PROGRAM progFCVCntrl
VAR
	FCV_04_0100 : fbFCV;
	FCV_04_1001 : fbFCV;
	FCV_04_1002 : fbFCV;
	FCV_04_1003 : fbFCV;
END_VAR

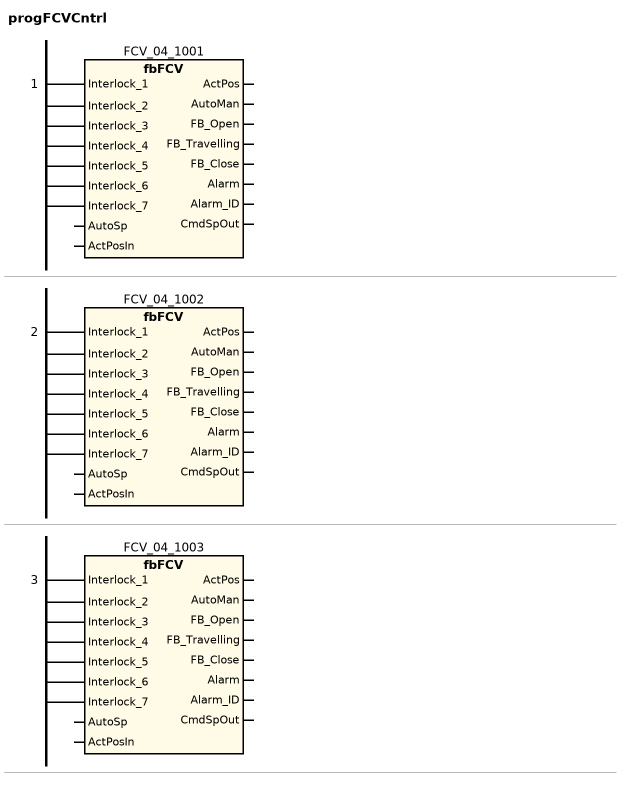
// NETWORK 1
FCV_04_1001(
    Interlock_1 := TRUE,
    Interlock_2 := TRUE,
    Interlock_3 := TRUE,
    Interlock_4 := TRUE,
    Interlock_5 := TRUE,
    Interlock_6 := TRUE,
    Interlock_7 := TRUE); // fbFCV

// NETWORK 2
FCV_04_1002(
    Interlock_1 := TRUE,
    Interlock_2 := TRUE,
    Interlock_3 := TRUE,
    Interlock_4 := TRUE,
    Interlock_5 := TRUE,
    Interlock_6 := TRUE,
    Interlock_7 := TRUE); // fbFCV

// NETWORK 3
FCV_04_1003(
    Interlock_1 := TRUE,
    Interlock_2 := TRUE,
    Interlock_3 := TRUE,
    Interlock_4 := TRUE,
    Interlock_5 := TRUE,
    Interlock_6 := TRUE,
    Interlock_7 := TRUE); // fbFCV

END_PROGRAM

(* stored: Version 1.1.0.1, ProductVersion 3.1.4022.17
   POU progFCVCntrl: Id {daadf6f8-5aa0-4fb6-94ed-3438b1933a51}, SpecialFunc None *)
